// TwinCAT 3 PLC project PLC1
// ProgramVersion: 3.1.4023.0
// libraries:
//   SimplePackML, * (Beckhoff Automation Poland)
//   Tc2_Standard, * (Beckhoff Automation GmbH)
//   Tc2_System, * (Beckhoff Automation GmbH)
//   Tc3_Module, * (Beckhoff Automation GmbH)
//   Tc3_PackML_V2, * (Beckhoff Automation GmbH)
// project tree:
//   / GlobalTextList.TcGTLO, PlcTask.TcTTO, Visualization Manager.TcVMO (not stored)
//   POUs/ FB_Conveyor.TcPOU, MAIN.TcPOU
//   VISUs/ Visualization.TcVIS
// real-time tasks:
//   TASK PlcTask: cycle T#10ms, priority 20, ADS port 350
//   TASK VISU_TASK: cycle T#200000us, priority 30, ADS port 351

CONFIGURATION PLC1
    RESOURCE PLC ON TwinCAT3
        TASK PlcTask(INTERVAL := T#10ms, PRIORITY := 20);
        PROGRAM MAIN WITH PlcTask : MAIN;
    END_RESOURCE
END_CONFIGURATION

// ---- POUs/MAIN.TcPOU
PROGRAM MAIN
VAR
	fbConveyor	: FB_Conveyor;
	sMode		: STRING;
END_VAR

fbConveyor(
	eModeCommand			:= , 
	eCommand				:= , 
	eMode					=> , 
	eState					=> , 
	bUndefinedDone			=> , 
	bInvalidModeCommandOut	=> , 
	bChangeIntoProduction	=> );
sMode := F_UnitModeToString(fbConveyor.eMode);

END_PROGRAM

// ---- POUs/FB_Conveyor.TcPOU
FUNCTION_BLOCK FB_Conveyor EXTENDS FB_Generic
VAR
	bExecuteComplete: BOOL;
	nStateChanges	: INT;
END_VAR

SUPER^();

{attribute 'object_name' := 'M_Execute'}
METHOD M_Execute
IF bExecuteComplete THEN
	bExecuteComplete := FALSE;
	M_StateComplete();
END_IF
END_METHOD

{attribute 'object_name' := 'M_Resetting'}
METHOD M_Resetting
VAR_INST
	delay	: TON;
END_VAR
delay( IN := NOT delay.Q, PT := T#2S );

IF delay.Q THEN
	THIS^.M_StateComplete();
END_IF
END_METHOD

{attribute 'object_name' := 'M_StateComplete'}
METHOD M_StateComplete
nStateChanges := nStateChanges + 1;
SUPER^.M_StateComplete();
END_METHOD

END_FUNCTION_BLOCK

// ---- GlobalTextList.TcGTLO
TEXTLIST GlobalTextList
  18 = 'Abort'
  33 = 'Aborted'
  34 = 'Aborting'
  16 = 'Clear'
  32 = 'Clearing'
  38 = 'Complete'
  39 = 'Completing'
  23 = 'Execute'
  25 = 'Held'
  12 = 'Hold'
  26 = 'Holding'
  21 = 'Idle'
  9 = 'Reset'
  30 = 'Reseting'
  36 = 'SC'
  10 = 'Start'
  22 = 'Starting'
  11 = 'Stop'
  31 = 'Stopped'
  35 = 'Stopping'
  14 = 'Suspend'
  28 = 'Suspended'
  29 = 'Suspending'
  13 = 'Unhold'
  24 = 'Unholding'
  37 = 'Unsuspend'
  27 = 'Unsuspending'
END_TEXTLIST

// ---- VISUs/Visualization.TcVIS
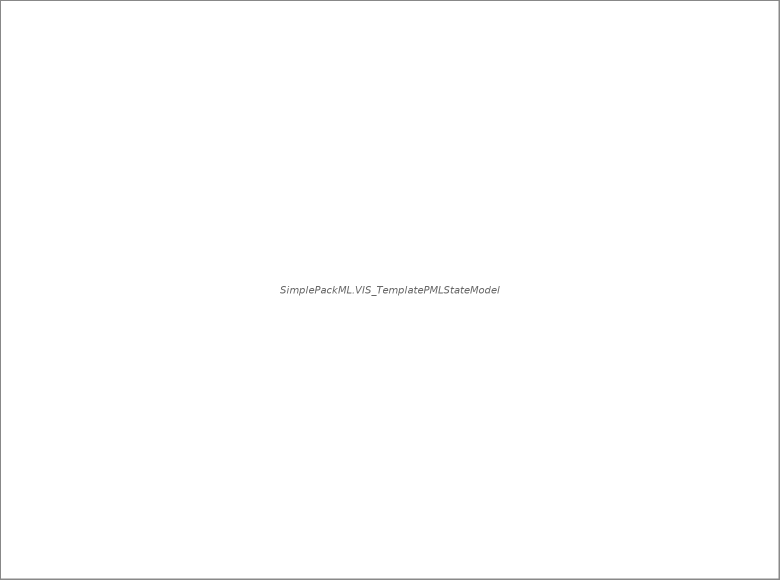
VISUALIZATION Visualization  // 780x580
    Frame (0,0 780x580)
        shows SimplePackML.VIS_TemplatePMLStateModel(ePMLUnitMode := MAIN.fbConveyor.eMode, ePMLState := MAIN.fbConveyor.eState)
END_VISUALIZATION
